(* IEC 61131-3 sources: PLC_DUAL_ORACLE/benchmark/tasks/medium/M05_conveyor_sequence, 1 file *)

(* ---- reference.st ---- *)
PROGRAM conveyor_seq
VAR_INPUT
    StartPB : BOOL;
    StopPB  : BOOL;
    EStop   : BOOL; (* normally-closed: TRUE = healthy, FALSE = activated *)
END_VAR
VAR_OUTPUT
    C1 : BOOL;
    C2 : BOOL;
END_VAR
VAR
    State : INT;
    T1    : TON;
END_VAR

(* Sequence delay runs while in Starting. T#2s = 2 scan ticks. *)
T1(IN := State = 1, PT := T#2s);

IF (NOT EStop) OR StopPB THEN
    State := 0;
ELSE
    CASE State OF
    0:
        IF StartPB THEN
            State := 1;
        END_IF;
    1:
        IF T1.Q THEN
            State := 2;
        END_IF;
    END_CASE;
END_IF;

CASE State OF
0:
    C1 := FALSE; C2 := FALSE;
1:
    C1 := FALSE; C2 := TRUE;
2:
    C1 := TRUE;  C2 := TRUE;
END_CASE;

END_PROGRAM
